Staubli VAL3: init.pgx

program init()
begin
  moveConfig = NOMINAL_CONFIG
  motionQueued = false
  reportEnabled = false
  reportInterval = 0.1
  selectedTool = endEffector
  target.config = ARM_CONFIG
end
